ABB RobotStudio station: Capstone.rsstnx

Station Capstone (saved by RobotStudio 23.4.10609.1)
Controller CRB15000_5_95
  mechanical unit ROB_1: CRB15000_5_95__02, 6 joints, base frame (0, 0, 0) mm
Layout (positions relative to the parent item):
  - CRB15000_5_95__02 [mechanism, from %ABB.RobotStudio.Models.CRB15000%\CRB15000_5_95__02.rslib] at (0, 0, 0) mm; joint values [0, -0.2386, 0.942, 0, -0.7033, 0] (rad or m)
  - Spreader [part] at (425.65, 0, 556.33) mm, size 150 x 100 x 10 mm
  - Part_2 [part] at (1000.05, -350, 160.84) mm, size 30 x 700 x 700 mm
Attachment: Spreader is attached to CRB15000_5_95__02 / Link6
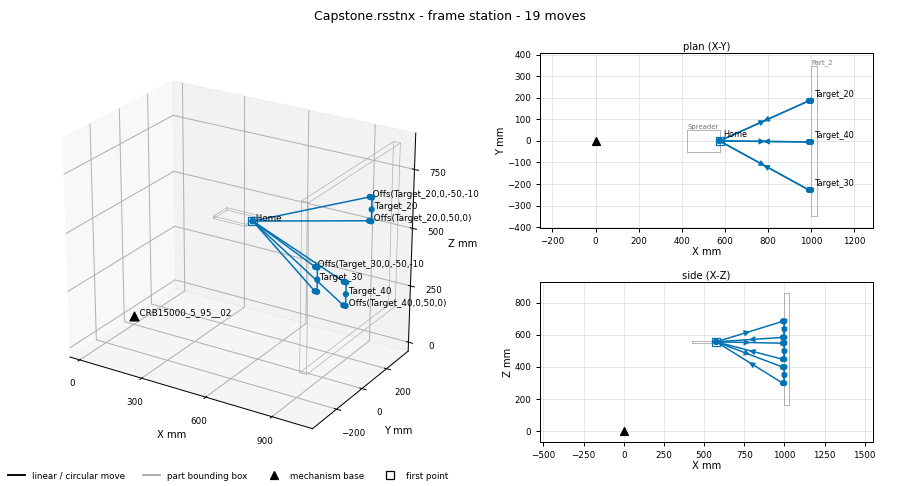
[picture p0: tool path of Capstone.rsstnx in frame station, 19 of 19 moves have a stored position in this frame; points joined in program order, loops and branches not executed]
Targets, tools, work objects and paths stored in the station, written as RAPID:
! task T_ROB1
MODULE CalibData
  TASK PERS tooldata SpreaderEOT:=[TRUE,[[0,0,150],[0.707106783,0.000000004,-0.000000001,-0.70710678]],[1,[0,0,1],[1,0,0,0],0,0,0]];
  TASK PERS wobjdata Wall:=[FALSE,TRUE,"",[[0,0,0],[1,0,0,0]],[[1000.052,350,860.843],[0.5,-0.5,0.5,-0.5]]];
ENDMODULE

! task T_ROB1
MODULE Module1
  CONST robtarget Target_10:=[[575.651830687,0.000001876,395.491214252],[0.499999995,-0.500000005,0.500000007,-0.499999993],[0,-1,0,1],[9E+09,9E+09,9E+09,9E+09,9E+09,9E+09]];
  CONST robtarget Target_20:=[[163.82,226.694,0],[0.965925826,0.258819045,0,0],[0,0,-1,1],[9E+09,9E+09,9E+09,9E+09,9E+09,9E+09]];
  CONST robtarget Target_30:=[[577.469,363.031,0],[0.965925826,0.258819045,0,0],[-1,-1,0,1],[9E+09,9E+09,9E+09,9E+09,9E+09,9E+09]];
  CONST robtarget Target_40:=[[354.533,512.021,0],[0.965925826,0.258819045,0,0],[-1,-1,0,1],[9E+09,9E+09,9E+09,9E+09,9E+09,9E+09]];
  CONST robtarget Home:=[[349.999998124,304.508785748,-424.400169313],[1,-0.000000012,0,0.000000002],[0,-1,0,1],[9E+09,9E+09,9E+09,9E+09,9E+09,9E+09]];
  PROC Path_10()
    MoveL Home,v1000,z100,SpreaderEOT\WObj:=Wall;
    MoveL Offs(Target_20,0,-50,-10),v1000,z100,SpreaderEOT\WObj:=Wall;
    MoveL Offs(Target_20,0,-50,0),v100,z100,SpreaderEOT\WObj:=Wall;
    MoveL Target_20,v100,z100,SpreaderEOT\WObj:=Wall;
    MoveL Offs(Target_20,0,50,0),v100,z100,SpreaderEOT\WObj:=Wall;
    MoveL Offs(Target_20,0,50,-10),v1000,z100,SpreaderEOT\WObj:=Wall;
    MoveL Home,v1000,z100,SpreaderEOT\WObj:=Wall;
    MoveL Offs(Target_30,0,-50,-10),v1000,z100,SpreaderEOT\WObj:=Wall;
    MoveL Offs(Target_30,0,-50,0),v100,z100,SpreaderEOT\WObj:=Wall;
    MoveL Target_30,v1000,z100,SpreaderEOT\WObj:=Wall;
    MoveL Offs(Target_30,0,50,0),v100,z100,SpreaderEOT\WObj:=Wall;
    MoveL Offs(Target_30,0,50,-10),v1000,z100,SpreaderEOT\WObj:=Wall;
    MoveL Home,v1000,z100,SpreaderEOT\WObj:=Wall;
    MoveL Offs(Target_40,0,-50,-10),v1000,z100,SpreaderEOT\WObj:=Wall;
    MoveL Offs(Target_40,0,-50,0),v100,z100,SpreaderEOT\WObj:=Wall;
    MoveL Target_40,v1000,z100,SpreaderEOT\WObj:=Wall;
    MoveL Offs(Target_40,0,50,0),v100,z100,SpreaderEOT\WObj:=Wall;
    MoveL Offs(Target_40,0,50,-10),v1000,z100,SpreaderEOT\WObj:=Wall;
    MoveL Home,v1000,z100,SpreaderEOT\WObj:=Wall;
  ENDPROC
  PROC main()
    Path_10;
  ENDPROC
ENDMODULE

! task T_ROB1
MODULE TorqueSensorCalib
  PROC TorqueSensorCal()
  ENDPROC
ENDMODULE

